PROGRAM git_Test
VAR
END_VAR

END_PROGRAM

(* stored: Version 1.1.0.1, ProductVersion 3.1.4024.12
   POU git_Test: Id {ff817349-10a0-05f9-0332-d8be63f4b9f3}, SpecialFunc None *)
